# EPICS autosave request: ADCore/ADApp/Db/NDFile_settings.req
$(P)$(R)FilePath
$(P)$(R)FileName
$(P)$(R)FileNumber
$(P)$(R)AutoIncrement
$(P)$(R)FileTemplate
$(P)$(R)AutoSave
$(P)$(R)FileFormat
$(P)$(R)FileWriteMode
$(P)$(R)NumCapture
$(P)$(R)DeleteDriverFile
